{attribute 'qualified_only'}
VAR_GLOBAL
    g_FastFaultOutput1  :   FB_HardwareFFOutput;	//FFO for Upstream Components
	g_fbArbiter1: FB_Arbiter(1);
END_VAR

(* stored: Version 1.1.0.1, ProductVersion 3.1.4022.18
   GVL GVL_PMPS: Id {0a30ac61-9bef-4090-bb2e-0e508084f744} *)
